# EPICS StreamDevice protocol: ort_994App/Db/ort_994.proto
#################################################
# ###                                       ### #
# ### StreamDevice Protocol for             ### #
# ### Ortec 994		                    ### #
# ###                                       ### #
# ### author: D. Hampai - M. Montis         ### #
# ###                                       ### #
# ### Ref 1.1; 2025-04-23                   ### #
#################################################

###################
# ### Globals ### #
###################

#Terminator = CR LF;
#Terminator = LF;
Terminator=CR;
ReplyTimeout=1000;
ReadTimeout=1000;
#HW_DEVICE="ortec";
DISP_UTIL="%s";
#
#	Protocols
#
##
#	Discard Extra Inputs
##
ExtraInput = Ignore;
#
getModel {
	out "SH_VER";
	in "%s";
}
setInit {
	out "INIT";
	in "%s";
        @init { out "INIT"; in "%s"; }
}
setDisplay {
        out "SET_DISP %s";
        in "%s";
        @init { out "SET_DISPLAY 0"; in "%s"; }
}
getSettings {
        out "SH_COU_PRE";
        in "%s";
}
setSettings {
        out "SET_COUNT_PRESET %s";
        in "%s";
        @init { out "SET_COUNT_PRESET 10,1"; in "%s"; }
}
setStop {
        out "STOP";
        in "%s";
}
getCount {
        out "SH_COU";
#	in "%8s;%8s;"
#        in "%(\$1)d;%(\$2)d;";
        in "%(\$1.B)d;%(\$1.C)d;";
}
clearCount {
        out "CL_COU";
        in "%s";
}
getDisplay {
        out "SH_DISP";
        in "$A00%{0245|1246}";
}
setStart {
	out "START";
	wait 1500;
	in "%s";
	out "STOP";
	in "%s";
}
#getReady {
#	out "1";
#}
